// TIA Portal V19 export
TYPE "LEXCHANGETRAY_typeNgStrapControlNode"
TITLE = exchangeTray_typeNgStrapControlNode
// exchangeTray_typeNgStrapControlNode related values
// stored: Access Published
   STRUCT
      commands { ExternalAccessible := 'False'; ExternalVisible := 'False'; ExternalWritable := 'False'} : "LEXCHANGETRAY_typeNgStrapControlNodeCommands";   // Module related commands from external systems
      monitoring { ExternalAccessible := 'False'; ExternalVisible := 'False'; ExternalWritable := 'False'} : "LEXCHANGETRAY_typeNgStrapContronNodeMonitoring";   // Module related monitoring information
   END_STRUCT;
END_TYPE
